(*~
    <docu>
        <summary>Sample component for inspiration</summary>
    </docu>
~*)
FUNCTION_BLOCK fbSampleComponent
VAR
    (*~
        <docu>
            <summary>Counter</summary>
            <remarks>
                > [!IMPORTANT]
                > This member is ignored when rendering.
            </remarks>
        </docu>
    ~*)
    {attribute clr [RenderIgnore()]}
    _counter : INT;
END_VAR
VAR
    (*~
        <docu>
            <summary>Counter</summary>
            <remarks>
                > [!IMPORTANT]
                > This member is readonly.
            </remarks>
        </docu>
    ~*)
    {attribute addProperty Name "Add Result"}
    {attribute clr [ReadOnly()]}
    _addResult : INT;
    {attribute addProperty Name "A"}
    _addNumberOne : INT;
    {attribute addProperty Name "B"}
    _addNumberTwo : INT;
END_VAR

(*~
    <docu>
        <summary>Adds two numbers</summary>
        <returns>Sum of two numbers</returns>
    </docu>
~*)
METHOD AddTwoNumbers : INT
VAR_INPUT
    NumberOne : INT;
    NumberTwo : INT;
END_VAR
AddTwoNumbers := NumberOne + NumberTwo;
END_METHOD

{attribute 'TcRpcEnable'}
METHOD INTERNAL AddTwoNumbersTest : INT
VAR_INPUT
    NumberOne : INT;
    NumberTwo : INT;
END_VAR
AddTwoNumbersTest := THIS^.AddTwoNumbers(NumberOne, NumberTwo);
END_METHOD

METHOD Cyclic
VAR_INPUT
END_VAR
_addResult := THIS^.AddTwoNumbers(_addNumberOne, _addNumberTwo);
END_METHOD

METHOD WaitForModulo : BOOL
VAR_INPUT
    Modulo : INT;
END_VAR
_counter := _counter + 1;
WaitForModulo := _counter MOD Modulo = 0;
END_METHOD

{attribute 'TcRpcEnable'}
METHOD INTERNAL WaitForModuloTest : BOOL
VAR_INPUT
    Modulo : INT;
END_VAR
WaitForModuloTest := THIS^.WaitForModulo(Modulo);
END_METHOD

END_FUNCTION_BLOCK

(* stored: Version 1.1.0.1, ProductVersion 3.1.4024.4
   POU fbSampleComponent: Id {58312ee6-e99b-4afb-aa9c-8c05761b5535}, SpecialFunc None
   Folder _tests: Id {5b8331b0-0029-4e78-a009-bf2eb8712373}
   Method AddTwoNumbers: Id {2ee747c8-6af4-41fb-afed-608159322163}
   Method AddTwoNumbersTest: Id {41574bed-82b4-4fb9-b188-7c2e9e506655}
   Method Cyclic: Id {bfe4b4a2-960e-417c-877e-2e6fa12b6282}
   Method WaitForModulo: Id {a1a1a029-7058-41f7-bac9-8a1faef1cdae}
   Method WaitForModuloTest: Id {be1c6e3d-fd9c-4e5d-a883-97b08c7f82b3} *)
